// This function has been automatically generated from the project information.
{attribute 'signature_flag' := '1073741824'}
{attribute 'TcGenerated'}
{attribute 'no-analysis'}
FUNCTION F_GetTitle : WSTRING
VAR_INPUT
	
END_VAR

F_GetTitle := "CNM_CycleManagerInterfaces";

END_FUNCTION

(* stored: Version 1.1.0.1
   POU F_GetTitle: Id {0b236df0-6ee7-4845-8720-6d4e7837b47e}, SpecialFunc None *)
